// TIA Portal V18 export
FUNCTION_BLOCK "p_trig_to_set_reset"   // FB38, FBD
{ S7_Optimized_Access := 'TRUE' }
VERSION : 0.1
// stored: AutoNumber true, IsIECCheckEnabled false, IsRetainMemResEnabled false, MemoryReserve 100, SetENOAutomatically false, UDAEnableTagReadback false
   VAR_INPUT
      "DO" : Bool;
   END_VAR
   VAR_OUTPUT
      DONE : Bool;
   END_VAR
   VAR_IN_OUT
      inout_button : Bool;
   END_VAR
   VAR
      mem_1 : Bool;
      mem_2 : Bool;
   END_VAR
   VAR_TEMP   // added for the SCL form of the ladder/FBD networks
      _w1 : Bool;
      _w2 : Bool;
   END_VAR
BEGIN

REGION Network 1
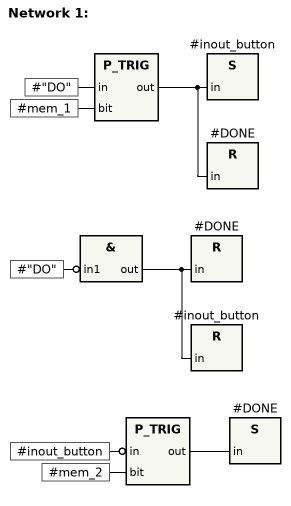
   #_w1 := #"DO" AND NOT #mem_1;   // rising edge
   #mem_1 := #"DO";
   IF #_w1 THEN
       #inout_button := TRUE;
       #DONE := FALSE;
   END_IF;
   IF NOT #"DO" THEN
       #DONE := FALSE;
       #inout_button := FALSE;
   END_IF;
   #_w2 := NOT #inout_button AND NOT #mem_2;   // rising edge
   #mem_2 := NOT #inout_button;
   IF #_w2 THEN #DONE := TRUE; END_IF;
END_REGION
END_FUNCTION_BLOCK
